(*
SPDX-FileCopyrightText: © 2026 Oleksandr Tiutyk <trofimich@gmail.com>
SPDX-License-Identifier: MIT
License: https://opensource.org/license/mit
*)

(*!
<summary>Captures the current library namespace through init_namespace.</summary>
<description>
The compiler initializes CurrentNamespace. The empty body requires no execution; consumers treat the output as
read-only metadata.
</description>
*)

FUNCTION_BLOCK INTERNAL NamespaceExtractor
VAR_OUTPUT
	//! <summary>Compiler-supplied library namespace; read-only to consumers.</summary>
	{attribute 'init_namespace'} 
	CurrentNamespace : STRING;	
END_VAR

END_FUNCTION_BLOCK

(* stored: Version 1.1.0.1
   POU NamespaceExtractor: Id {31b409a2-9b59-4c74-8400-c96623e521ca}, SpecialFunc None *)
